(* PLC project CoDeSys External Library Template, WAGO e!COCKPIT e!COCKPIT, author 3S - Smart Software Solutions GmbH *)
(* stored: creationDateTime 2019-10-29T12:37:19.7708223, version 3.5.5.30, modificationDateTime 2019-10-29T12:36:39.3744516, organization 3S - Smart Software Solutions GmbH *)
(* Library project template with all possible element types, docu and a sample project structure *)

FUNCTION fnCRC16Odbieranie : BOOL
  VAR_INPUT
    arReceiverBuffer : ARRAY[1..512] OF BYTE;
    udiRxNBytes : UDINT;
    sMACAdresAplikacji : STRING;
    abMACAdresAplikacji : ARRAY[1..6] OF BYTE;
  END_VAR
  VAR_IN_OUT
    sKomunikat : alSTRINGKomunikat;
  END_VAR
  VAR
    wCRC16_modbus : WORD;
    intPetla : INT;
    arwTelegram : ARRAY[1..512] OF BYTE;
  END_VAR

            wCRC16_modbus := MEM.CRC16_modbus(ADR(arReceiverBuffer[1]) , UDINT_TO_UINT(udiRxNBytes) - 2);
sKomunikat := '';
IF (MEM.LowByte(wCRC16_modbus) = arReceiverBuffer[udiRxNBytes - 1] AND MEM.HighByte(wCRC16_modbus) = arReceiverBuffer[udiRxNBytes]) OR ASCIIByte_to_string(arReceiverBuffer[1]) = 'Z' THEN
	fnCRC16Odbieranie := TRUE;
	FOR intPetla := 1 TO (UDINT_TO_INT(udiRxNBytes) - 2) BY 1 DO
		IF intPetla >= 7 AND intPetla <= 12 AND arReceiverBuffer[7] = abMACAdresAplikacji[1] AND arReceiverBuffer[8] = abMACAdresAplikacji[2] AND arReceiverBuffer[9] = abMACAdresAplikacji[3] AND 
			arReceiverBuffer[10] = abMACAdresAplikacji[4] AND arReceiverBuffer[11] = abMACAdresAplikacji[5] AND arReceiverBuffer[12] = abMACAdresAplikacji[6] THEN
			sKomunikat := CONCAT(sKomunikat , MID(sMACAdresAplikacji, 1 , intPetla - 6));
		ELSE
			sKomunikat := CONCAT(sKomunikat , ASCIIByte_to_string(arReceiverBuffer[intPetla]));
		END_IF
	END_FOR
	ELSE
	fnCRC16Odbieranie := FALSE;	
END_IF

          
END_FUNCTION
